(* CODESYS project Reporte2.project

Project tree, tasks and I/O mapping:
  Device : CECC-LK, Festo AG & Co. KG, order no. 574418, version 3.5.3.1
    application Application
      libraries: Standard, 3.5.15.0 (System)
      task MainTask (cyclic, interval t#20ms, priority 20) calls nothing
      program PLC_PRG [LD]
      visualisation Visualization
    Onboard : CECC 14I/8O, Festo AG & Co. KG, version 3.4.5.5
        unmapped channels: Onboard Input, Onboard Output
      Digital Inputs
          unmapped channels: Onboard Input
      Digital Outputs
          unmapped channels: Onboard Output
  text list GlobalTextList
*)

// Device/Application/PLC_PRG
PROGRAM PLC_PRG
VAR
	S1: BOOL;
	B1: BOOL;
	Y1: BOOL;
	B2: BOOL;
END_VAR

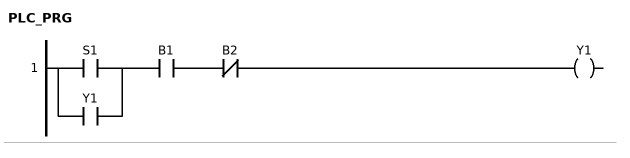
// NETWORK 1
Y1 := (S1 OR Y1) AND B1 AND NOT B2;

END_PROGRAM

// Device/Application/Visualization
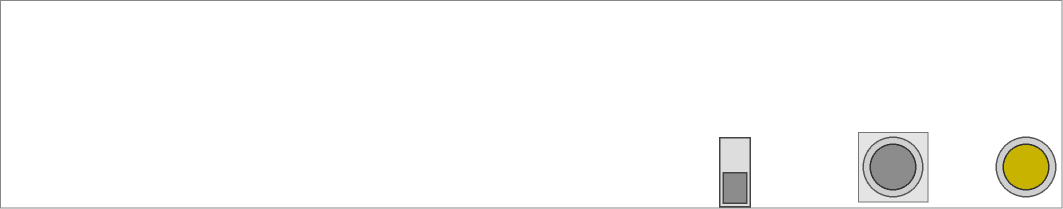
VISUALIZATION Visualization  // 1063x209
    DipSwitch (700,137 70x70), variable: PLC_PRG.S1, behaviour: TOGGLE, style: Switch-DipSwitch-Gray
    PushSwitch (858,132 70x70), variable: PLC_PRG.B1, behaviour: TOGGLE, style: Switch-PushSwitch-Gray
    Lamp1 (991,132 70x70), variable: PLC_PRG.Y1, style: Lamp-Lamp1-Yellow
END_VISUALIZATION
